Omron Sysmac Studio project nx1p2_ss_5 (Sysmac Studio 1.45.1.64010, StandardProject)

# Controller new_Controller_0: NX1P2-9024DT version 1.40
Units and slaves: Node86 : NX-ECC201 (E001); Unit 1 : NX-OD5121 (N1); Unit 2 : NX-OD4256 (N2); Unit 3 : NX-ID5342 (N3); Unit 4 : NX-ID5442 (N4); Node1 : GX-ID1611+OD16 (E002)
Task PrimaryTask (priority 4, period or condition 2000): Program0

VAR_GLOBAL
    NX1P2_OUT_0 : BOOL;  (* INPUT_NX1P2; at BuiltInIO://cpu/#0/Output_Bit_00 *)
    NX1P2_OUT_1 : BOOL;  (* INPUT_NX1P2; at BuiltInIO://cpu/#0/Output_Bit_01 *)
    NX1P2_OUT_2 : BOOL;  (* INPUT_NX1P2; at BuiltInIO://cpu/#0/Output_Bit_02 *)
    NX1P2_OUT_3 : BOOL;  (* INPUT_NX1P2; at BuiltInIO://cpu/#0/Output_Bit_03 *)
    NX1P2_OUT_4 : BOOL;  (* INPUT_NX1P2; at BuiltInIO://cpu/#0/Output_Bit_04 *)
    NX1P2_OUT_5 : BOOL;  (* INPUT_NX1P2; at BuiltInIO://cpu/#0/Output_Bit_05 *)
    NX1P2_OUT_6 : BOOL;  (* INPUT_NX1P2; at BuiltInIO://cpu/#0/Output_Bit_06 *)
    NX1P2_OUT_7 : BOOL;  (* INPUT_NX1P2; at BuiltInIO://cpu/#0/Output_Bit_07 *)
    NX1P2_OUT_8 : BOOL;  (* INPUT_NX1P2; at BuiltInIO://cpu/#0/Output_Bit_08 *)
    NX1P2_OUT_9 : BOOL;  (* INPUT_NX1P2; at BuiltInIO://cpu/#0/Output_Bit_09 *)
    NX1P2_IN_0 : BOOL;  (* NX1P2_INPUT; at BuiltInIO://cpu/#0/Input_Bit_00 *)
    NX1P2_IN_1 : BOOL;  (* NX1P2_INPUT; at BuiltInIO://cpu/#0/Input_Bit_01 *)
    NX1P2_IN_2 : BOOL;  (* NX1P2_INPUT; at BuiltInIO://cpu/#0/Input_Bit_02 *)
    NX1P2_IN_3 : BOOL;  (* NX1P2_INPUT; at BuiltInIO://cpu/#0/Input_Bit_03 *)
    NX1P2_IN_4 : BOOL;  (* NX1P2_INPUT; at BuiltInIO://cpu/#0/Input_Bit_04 *)
    NX1P2_IN_5 : BOOL;  (* NX1P2_INPUT; at BuiltInIO://cpu/#0/Input_Bit_05 *)
    NX1P2_IN_6 : BOOL;  (* NX1P2_INPUT; at BuiltInIO://cpu/#0/Input_Bit_06 *)
    NX1P2_IN_7 : BOOL;  (* NX1P2_INPUT; at BuiltInIO://cpu/#0/Input_Bit_07 *)
    NX1P2_IN_8 : BOOL;  (* NX1P2_INPUT; at BuiltInIO://cpu/#0/Input_Bit_08 *)
    NX1P2_IN_9 : BOOL;  (* NX1P2_INPUT; at BuiltInIO://cpu/#0/Input_Bit_09 *)
    NX1P2_IN_10 : BOOL;  (* NX1P2_INPUT; at BuiltInIO://cpu/#0/Input_Bit_10 *)
    NX1P2_IN_11 : BOOL;  (* NX1P2_INPUT; at BuiltInIO://cpu/#0/Input_Bit_11 *)
    NX1P2_IN_12 : BOOL;  (* NX1P2_INPUT; at BuiltInIO://cpu/#0/Input_Bit_12 *)
    NX1P2_IN_13 : BOOL;  (* NX1P2_INPUT; at BuiltInIO://cpu/#0/Input_Bit_13 *)
    OD5121_OUT_0 : BOOL;  (* OD5121; at ECAT://node#[86,1]/Output Bit 16 bits/Output Bit 00 *)
    OD5121_OUT_1 : BOOL;  (* OD5121; at ECAT://node#[86,1]/Output Bit 16 bits/Output Bit 01 *)
    OD5121_OUT_2 : BOOL;  (* OD5121; at ECAT://node#[86,1]/Output Bit 16 bits/Output Bit 02 *)
    OD5121_OUT_3 : BOOL;  (* OD5121; at ECAT://node#[86,1]/Output Bit 16 bits/Output Bit 03 *)
    OD5121_OUT_4 : BOOL;  (* OD5121; at ECAT://node#[86,1]/Output Bit 16 bits/Output Bit 04 *)
    OD5121_OUT_5 : BOOL;  (* OD5121; at ECAT://node#[86,1]/Output Bit 16 bits/Output Bit 05 *)
    OD5121_OUT_6 : BOOL;  (* OD5121; at ECAT://node#[86,1]/Output Bit 16 bits/Output Bit 06 *)
    OD5121_OUT_7 : BOOL;  (* OD5121; at ECAT://node#[86,1]/Output Bit 16 bits/Output Bit 07 *)
    OD5121_OUT_8 : BOOL;  (* OD5121; at ECAT://node#[86,1]/Output Bit 16 bits/Output Bit 08 *)
    OD5121_OUT_9 : BOOL;  (* OD5121; at ECAT://node#[86,1]/Output Bit 16 bits/Output Bit 09 *)
    OD5121_OUT_10 : BOOL;  (* OD5121; at ECAT://node#[86,1]/Output Bit 16 bits/Output Bit 10 *)
    OD5121_OUT_11 : BOOL;  (* OD5121; at ECAT://node#[86,1]/Output Bit 16 bits/Output Bit 11 *)
    OD5121_OUT_12 : BOOL;  (* OD5121; at ECAT://node#[86,1]/Output Bit 16 bits/Output Bit 12 *)
    OD5121_OUT_13 : BOOL;  (* OD5121; at ECAT://node#[86,1]/Output Bit 16 bits/Output Bit 13 *)
    OD5121_OUT_14 : BOOL;  (* OD5121; at ECAT://node#[86,1]/Output Bit 16 bits/Output Bit 14 *)
    OD5121_OUT_15 : BOOL;  (* OD5121; at ECAT://node#[86,1]/Output Bit 16 bits/Output Bit 15 *)
    OD5121_REGISTER : WORD;  (* OD5121; at ECAT://node#[86,1]/Output Bit 16 bits *)
    OD4256_OUT_0 : BOOL;  (* OD4256; at ECAT://node#[86,2]/Output Bit 8 bits/Output Bit 00 *)
    OD4256_OUT_1 : BOOL;  (* OD4256; at ECAT://node#[86,2]/Output Bit 8 bits/Output Bit 01 *)
    OD4256_OUT_2 : BOOL;  (* OD4256; at ECAT://node#[86,2]/Output Bit 8 bits/Output Bit 02 *)
    OD4256_OUT_3 : BOOL;  (* OD4256; at ECAT://node#[86,2]/Output Bit 8 bits/Output Bit 03 *)
    OD4256_OUT_4 : BOOL;  (* OD4256; at ECAT://node#[86,2]/Output Bit 8 bits/Output Bit 04 *)
    OD4256_OUT_5 : BOOL;  (* OD4256; at ECAT://node#[86,2]/Output Bit 8 bits/Output Bit 05 *)
    OD4256_OUT_6 : BOOL;  (* OD4256; at ECAT://node#[86,2]/Output Bit 8 bits/Output Bit 06 *)
    OD4256_OUT_7 : BOOL;  (* OD4256; at ECAT://node#[86,2]/Output Bit 8 bits/Output Bit 07 *)
    OD4256_REGISTER : BYTE;  (* OD4256; at ECAT://node#[86,2]/Output Bit 8 bits *)
    GX_OUT_0 : BOOL;  (* GX_WXT_OD16 *)
    GX_OUT_1 : BOOL;  (* GX_WXT_OD16 *)
    GX_OUT_2 : BOOL;  (* GX_WXT_OD16 *)
    GX_OUT_3 : BOOL;  (* GX_WXT_OD16 *)
    GX_OUT_4 : BOOL;  (* GX_WXT_OD16 *)
    GX_OUT_5 : BOOL;  (* GX_WXT_OD16 *)
    GX_OUT_6 : BOOL;  (* GX_WXT_OD16 *)
    GX_OUT_7 : BOOL;  (* GX_WXT_OD16 *)
    GX_OUT_8 : BOOL;  (* GX_WXT_OD16 *)
    GX_OUT_9 : BOOL;  (* GX_WXT_OD16 *)
    GX_OUT_10 : BOOL;  (* GX_WXT_OD16 *)
    GX_OUT_11 : BOOL;  (* GX_WXT_OD16 *)
    GX_OUT_12 : BOOL;  (* GX_WXT_OD16 *)
    GX_OUT_13 : BOOL;  (* GX_WXT_OD16 *)
    GX_OUT_14 : BOOL;  (* GX_WXT_OD16 *)
    GX_OUT_15 : BOOL;  (* GX_WXT_OD16 *)
    REGISTER_GX_OUT : WORD;  (* GX_WXT_OD16 *)
    IN_GX_0 : BOOL;  (* INPUT_GX_ID_1611 *)
    IN_GX_1 : BOOL;  (* INPUT_GX_ID_1611 *)
    IN_GX_2 : BOOL;  (* INPUT_GX_ID_1611 *)
    IN_GX_3 : BOOL;  (* INPUT_GX_ID_1611 *)
    IN_GX_4 : BOOL;  (* INPUT_GX_ID_1611 *)
    IN_GX_5 : BOOL;  (* INPUT_GX_ID_1611 *)
    IN_GX_6 : BOOL;  (* INPUT_GX_ID_1611 *)
    IN_GX_7 : BOOL;  (* INPUT_GX_ID_1611 *)
    IN_GX_8 : BOOL;  (* INPUT_GX_ID_1611 *)
    IN_GX_9 : BOOL;  (* INPUT_GX_ID_1611 *)
    IN_GX_10 : BOOL;  (* INPUT_GX_ID_1611 *)
    IN_GX_11 : BOOL;  (* INPUT_GX_ID_1611 *)
    IN_GX_12 : BOOL;  (* INPUT_GX_ID_1611 *)
    IN_GX_13 : BOOL;  (* INPUT_GX_ID_1611 *)
    IN_GX_14 : BOOL;  (* INPUT_GX_ID_1611 *)
    IN_GX_15 : BOOL;  (* INPUT_GX_ID_1611 *)
    REGISTER_IN_GX : WORD;  (* INPUT_GX_ID_1611 *)
    ERROR_GX : BYTE;  (* INPUT_GX_ID_1611 *)
END_VAR

PROGRAM Program0
VAR
    m0 : BOOL;
    M1 : BOOL;
END_VAR
VAR_EXTERNAL
    NX1P2_IN_0 : BOOL;
    NX1P2_OUT_0 : BOOL;
END_VAR

(* Section Section0: ladder, written here as Structured Text *)

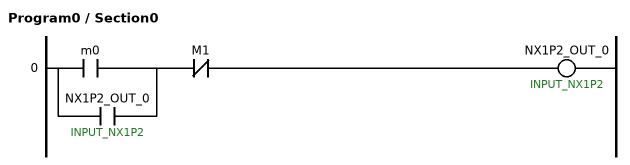
(* Rung 0 *)
NX1P2_OUT_0 := (m0 OR NX1P2_OUT_0) AND NOT M1;
END_PROGRAM